// TIA Portal V19 export
VAR_GLOBAL   // PLC tag table "Digitale Ausgänge"
   A_Dkl_li_auf_CM01 AT %Q0.0 : Bool;   // Deckel links öffnen Säure CM01
   A_Dkl_li_zu_CM01 AT %Q0.1 : Bool;   // Deckel links schließen Säure CM01
   A_Dkl_re_auf_CM01 AT %Q0.2 : Bool;   // Deckel rechts öffnen Säure CM01
   A_Dkl_re_zu_CM01 AT %Q0.3 : Bool;   // Deckel rechts schließen Säure CM01
   A_Dkl_li_auf_CM02 AT %Q0.4 : Bool;   // Deckel links öffnen Säure CM02
   A_Dkl_li_zu_CM02 AT %Q0.5 : Bool;   // Deckel links schließen Säure CM02
   A_Dkl_re_auf_CM02 AT %Q0.6 : Bool;   // Deckel rechts öffnen Säure CM02
   A_Dkl_re_zu_CM02 AT %Q0.7 : Bool;   // Deckel rechts schließen Säure CM02
   "R A 1.0" AT %Q1.0 : Bool;   // Reserve
   A_LED_Q_Err AT %Q1.1 : Bool;   // LED in Taster Fehlerquittung
   A_LED_Q_NH AT %Q1.2 : Bool;   // LED in NOT-HALT Quittung
   "R A 1.3" AT %Q1.3 : Bool;   // Reserve
   "R A1.4" AT %Q1.4 : Bool;   // Turmleuchte Reserve Be-/Entladestation
   A_Mld_fertig AT %Q1.5 : Bool;   // Meldung fertig
   A_Mld_Automatik AT %Q1.6 : Bool;   // Meldung Automatik
   A_Mld_Wrn AT %Q1.7 : Bool;   // Meldung Warnung
   A_Mld_Al AT %Q2.0 : Bool;   // Meldung Störung
   A_Hupe AT %Q2.1 : Bool;   // Hupe
   A_TL_T_Vorarlarm_Gas AT %Q2.7 : Bool;   // Voralarm Gas (E13.2.)TL Tür
   A_TL_T_Hauptalarm_Gas AT %Q3.0 : Bool;   // Hauptalarm Gas (13.3) TL Tür
   A_TL_T_Hupe AT %Q3.1 : Bool;   // Hupe TL Tür
   A_KS_CM05_nicht_Voll AT %Q3.2 : Bool;   // Meldung an Wäscher Sammeltank CM05 voll
   A_KS_in_Betrieb AT %Q3.3 : Bool;   // Meldung an Wäscher und Neutralisation Säureanlage in Betrieb
   A_Mld_WS_Leckage AT %Q3.4 : Bool;   // Meldung an Werkschutz Leckage
   A_Mld_WS_Ueberlauf AT %Q3.5 : Bool;   // Meldung an Werkschutz Überlauf
   A_Mld_WS_SSt AT %Q3.6 : Bool;   // Meldung an Werkschutz Sammelstörung
   "R A 3.7" AT %Q3.7 : Bool;   // digitaler Ausgang Reserve Neutralisation
   "R A 4.0" AT %Q4.0 : Bool;   // digitaler Ausgang Reserve 1
   "R A 4.1" AT %Q4.1 : Bool;   // digitaler Ausgang Reserve 2
   "R A 4.2" AT %Q4.2 : Bool;   // digitaler Ausgang Reserve 3
   "A_Mld_fertig_Geb.G" AT %Q4.3 : Bool;   // Meldung fertig A_Mld_Automatik
   A_LED_Tuer_VS AT %Q6.0 : Bool;   // LED Tür Vorderseite CL02.SF17
   A_LED_Tuer_RS AT %Q6.1 : Bool;   // LED Tür Rückseite CL02.SF18
   A_Frg_FU_FP_HQ01 AT %Q6.2 : Bool;   // Freigabe FP HQ01 Säure CM01 CM01.GP01
   A_Frg_FU_UP_HF_CM01 AT %Q6.3 : Bool;   // Freigabe UWP Säure CM01 CM01.GP02
   A_Frg_FU_UP_H2O_CM03 AT %Q6.4 : Bool;   // Freigabe UWP Spüle CM03 CM03.GP03
   A_Frg_FU_FP_HQ02 AT %Q6.5 : Bool;   // Freigabe FP HQ02 Säure CM02 CM02.GP04
   A_Frg_FU_UP_HF_CM02 AT %Q6.6 : Bool;   // Freigabe UWP Säure CM02 CM02.GP05
   A_Frg_FU_UP_H2O_CM04 AT %Q6.7 : Bool;   // Freigabe UWP Spüle CM04 CM04.GP06
   A_Frg_FU_Vent AT %Q7.0 : Bool;   // Ventilator Ein Sperrluft FP02.GQ01
   A_RT_auf AT %Q7.1 : Bool;   // Schnelllauftor öffnen Ein-/Ausfahrt
   A_RT_zu AT %Q7.2 : Bool;   // Schnelllauftor schließen Ein-/Ausfahrt
   A_Pu_Entl_CM05 AT %Q7.3 : Bool;   // Pumpe Ein Entleerung Sammeltank CM05.GP11
   "R A 5.4" AT %Q5.4 : Bool;
   "R A 5.5" AT %Q5.5 : Bool;
   "R A 5.6" AT %Q5.6 : Bool;
   "R A 5.7" AT %Q5.7 : Bool;
   "R A 7.4" AT %Q7.4 : Bool;
   "R A 7.5" AT %Q7.5 : Bool;
   "R A 7.6" AT %Q7.6 : Bool;
   "R A 7.7" AT %Q7.7 : Bool;
   A_IBC_Vers AT %Q32.0 : Bool;   // IBC vorhanden Versorgung
   "R A 32.1" AT %Q32.1 : Bool;   // Reserve gelb Versorgung
   "R A 32.2" AT %Q32.2 : Bool;   // Reserve rot Versorgung
   "R A 32.3" AT %Q32.3 : Bool;   // Reserve Hupe Versorgung
   A_IBC_Ents AT %Q32.4 : Bool;   // IBC vorhanden Entsorgung
   "R A 32.5" AT %Q32.5 : Bool;   // Reserve gelb Versorgung
   "R A 32.6" AT %Q32.6 : Bool;   // Reserve rot Versorgung
   "R A 32.7" AT %Q32.7 : Bool;   // Reserve Hupe Versorgung
   "R A 33.0" AT %Q33.0 : Bool;
   "R A 33.1" AT %Q33.1 : Bool;
   "R A 33.2" AT %Q33.2 : Bool;
   "R A 33.3" AT %Q33.3 : Bool;
   "R A 33.4" AT %Q33.4 : Bool;
   "R A 33.5" AT %Q33.5 : Bool;
   "R A 33.6" AT %Q33.6 : Bool;
   "R A 33.7" AT %Q33.7 : Bool;
   "A_CM01.QM18" AT %Q48.0 : Bool;   // Eingang Saugleitung Filterpumpe GP01 Säure 01 CM01.QM18
   "A_CM01.QM19" AT %Q48.1 : Bool;   // Eingang Spülleitung Filterpumpe GP01 Säure 01 CM01.QM19
   "A_CM01.QM20" AT %Q48.2 : Bool;   // Eingang Spülleitung Umwälzpumpe GP02 Säure 01 CM01.QM20
   "A_HQ01.QM21" AT %Q48.4 : Bool;   // Eingang SäureleitungFiltereinheit HQ01Säure 01HQ01.QM21
   "A_HQ01.LV01" AT %Q48.3 : Bool;   // Entlüftungs-/ Überdruckventil Beutelfilter Säure 01 HQ01.LV01
   "A_HQ01.QM22" AT %Q48.5 : Bool;   // Eingang Spülleitung Filtereinheit HQ01 Säure 01 HQ01.QM22
   "A_HQ01.QM23" AT %Q48.6 : Bool;   // Ausgang Säureleitung Filtereinheit HQ01 Säure 01 HQ01.QM23
   "A_HQ01.QM24" AT %Q48.7 : Bool;   // Ausgang Spülleitung Filtereinheit HQ01 Säure 01 zu Sammeltank HQ01.QM24
   "A_CM01.QM25" AT %Q49.0 : Bool;   // Eingang Saugleitung Umwälzpumpe GP02 Säure 01 CM01.QM25
   "A_CM01.QM26" AT %Q49.1 : Bool;   // Ausgang Druckleitung Umwälzpumpe GP02 Säure 01 CM01.QM26
   "A_CM01.QM27" AT %Q49.2 : Bool;   // Ausgang Spülleitung Umwälzpumpe GP02 Säure 01 zu Sammeltank CM01.QM27
   "A_CM03.QM33" AT %Q49.3 : Bool;   // Eingang Saugleitung Umwälzpumpe GP03 Spülbecken 1 CM03.QM33
   "A_CM03.QM34" AT %Q49.4 : Bool;   // Ausgang Druckleitung Umwälzpumpe GP03 Spülbecken 1 CM03.QM34
   "A_CM03.QM36" AT %Q49.5 : Bool;   // Eingang Spülleitung Umwälzpumpe GP03 Spülbecken 1 CM03.QM36
   "A_CM03.QM37" AT %Q49.6 : Bool;   // Ausgang Spülleitung Umwälzpumpe GP03 Spülbecken 1 CM03.QM37
   "R A 49.7" AT %Q49.7 : Bool;   // Magnetventil Reserve
   "A_CM02.QM55" AT %Q50.0 : Bool;   // Eingang Saugleitung Filterpumpe GP04 Säure 02 CM02.QM55
   "A_CM02.QM56" AT %Q50.1 : Bool;   // Eingang Spülleitung Filterpumpe GP04 Säure 02 CM02.QM56
   "A_CM02.QM57" AT %Q50.2 : Bool;   // Eingang Spülleitung Umwälzpumpe GP05 Säure 02 CM02.QM57
   "A_HQ02.QM58" AT %Q50.4 : Bool;   // Eingang Spülleitung Filtereinheit HQ02 Säure 02 HQ02.QM58
   "A_HQ02.LV02" AT %Q50.3 : Bool;   // Entlüftungs-/ Überdruckventil Beutelfilter Säure 02 HQ02.LV02
   "A_HQ02.QM59" AT %Q50.5 : Bool;   // Eingang Säureleitung Filtereinheit HQ02 Säure 02 HQ02.QM59
   "A_HQ02.QM60" AT %Q50.6 : Bool;   // Ausgang Säureleitung Filtereinheit HQ02 Säure 02 HQ02.QM60
   "A_HQ02.QM61" AT %Q50.7 : Bool;   // Ausgang Spülleitung Filtereinheit HQ02 Säure 02 zu Sammeltank HQ02.QM61
   "A_CM02.QM62" AT %Q51.0 : Bool;   // Eingang Saugleitung Umwälzpumpe GP05 Säure 02 CM02.QM62
   "A_CM02.QM63" AT %Q51.1 : Bool;   // Ausgang Druckleitung Umwälzpumpe GP05 Säure 02 CM02.QM63
   "A_CM02.QM64" AT %Q51.2 : Bool;   // Ausgang Spülleitung Umwälzpumpe GP05 Säure 02 zu Sammeltank CM02.QM64
   "R A 51.3" AT %Q51.3 : Bool;   // Magnetventil Reserve
   "A_CM04.QM72" AT %Q51.4 : Bool;   // Eingang Saugleitung Umwälzpumpe GP06 Spülbecken 2 CM04.QM72
   "A_CM04.QM73" AT %Q51.5 : Bool;   // Ausgang Druckleitung Umwälzpumpe GP06 Spülbecken 2 CM04.QM73
   "A_CM04.QM75" AT %Q51.6 : Bool;   // Eingang Spülleitung Umwälzpumpe GP06 Spülbecken 2 CM04.QM75
   "R A 51.7" AT %Q51.7 : Bool;   // Magnetventil Reserve
   "A_CM04.QM76" AT %Q52.0 : Bool;   // Ausgang Spülleitung Umwälzpumpe GP06 Spülbecken 2 CM04.QM76
   "A_CM04.QM77" AT %Q52.1 : Bool;   // Frischwasserzufuhr Nachdosierung Spülbecken 2 CM04.QM77
   "A_CL01.GP08" AT %Q52.2 : Bool;   // Membranpumpe GP08 Sumpfentleerung Übergabestation CL01.GP08
   "A_CL02.GP09" AT %Q52.3 : Bool;   // Membranpumpe GP09 Sumpfentleerung Säurebecken CL02.GP09
   "A_CL01.QM51" AT %Q52.4 : Bool;   // Zuleitung VE-Wasser-Spülung Pumpe GP08 CL01.QM51
   "A_CL02.QM52" AT %Q52.5 : Bool;   // Zuleitung VE-Wasser-Spülung Pumpe GP09 CL01.QM52
   "R A 52.6" AT %Q52.6 : Bool;   // Magnetventil Reserve
   "R A 52.7" AT %Q52.7 : Bool;   // Magnetventil Reserve
   "A_CM05.QM61" AT %Q53.0 : Bool;   // Saugseite Förderpumpe Entleerung GP11 Sammeltank CM05 CM05.QM61
   "A_CM05.QM62" AT %Q53.1 : Bool;   // Eingang Spülleitung Förderpumpe GP11 Sammeltank CM05 CM05.QM62
   "A_CM05.QM63" AT %Q53.2 : Bool;   // Ausgang Spülleitung Förderpumpe GP11 Sammeltank CM05 CM05.QM63
   "A_CM05.QM64" AT %Q53.3 : Bool;   // Druckseite Förderpumpe Entleerung GP11 Sammeltank CM05 CM05.QM64
   "R A 53.4" AT %Q53.4 : Bool;   // Magnetventil Reserve
   "R A 53.5" AT %Q53.5 : Bool;   // Magnetventil Reserve
   "R A 53.6" AT %Q53.6 : Bool;   // Magnetventil Reserve
   "R A 53.7" AT %Q53.7 : Bool;   // Magnetventil Reserve
   "A_CM03.QM35" AT %Q64.0 : Bool;   // VE-Wasserleitung Spritzregister Spülbecken 1 CM03.QM35
   "A_CM04.QM74" AT %Q64.1 : Bool;   // VE-Wasserleitung Spritzregister Spülbecken 2 CM04.QM74
   "A_GP01.GP12" AT %Q64.2 : Bool;   // Druckluftmembran- Leckagepumpe GP12 Versorgung Frischsäure GP01.GP12
   "A_GP01.GP13" AT %Q64.3 : Bool;   // Druckluftmembran- pumpe GP13 Versorgung Frischsäure GP01.GP13
   "A_GP01.QM14" AT %Q64.4 : Bool;   // PFA Schlauchleitung Anbindung IBC Quick Connect Entsorgung GP01.QM14
   "A_GP01.QM15" AT %Q64.5 : Bool;   // Eingang Saugleitung Membranpumpe GP13 Versorgung Frischsäure GP01.QM15
   "A_GP01.QM16" AT %Q64.6 : Bool;   // Eingang Spülleitung Membranpumpe GP13 Versorgung Frischsäure GP01.QM16
   "A_GP01.QM17" AT %Q64.7 : Bool;   // Ausgang Spülleitung Membranpumpe GP13 Versorgung zu Sammeltank GP01.QM17
   "A_GP01.QM18" AT %Q65.0 : Bool;   // Ausgang Druckleitung Membranpumpe GP13 Versorgung zu UV-GP01 GP01.QM18
   "A_GP01.QM19" AT %Q65.1 : Bool;   // Verriegelung UV-GP01 Versorgungsleitung zu Säure CM02 GP01.QM19
   "A_GP01.QM20" AT %Q65.2 : Bool;   // Verriegelung UV-GP01 Versorgungsleitung zu Säure CM01 GP01.QM20
   "A_GP01.QM21" AT %Q65.3 : Bool;   // Verriegelung UV-GP01 Versorgungsleitung zur Entsorgung GP02 GP01.QM21
   "A_GP01.QM22" AT %Q65.4 : Bool;   // Verriegelung UV-GP01 Versorgungsleitung zur Versorgung GP01 GP01.QM22
   "A_GP01.QM23" AT %Q65.5 : Bool;   // VE-Wasser-Spülung GP12 zu Auffangwanne GP01.QM23
   "A_GP02.GP07" AT %Q65.6 : Bool;   // Druckluftmembran- Leckagepumpe GP07 Entsorgung Altsäure GP02.GP07
   "A_GP02.GP10" AT %Q65.7 : Bool;   // Druckluftmembran- pumpe GP10 Versorgung aus GP02 GP02.GP10
   "A_GP02.QM37" AT %Q66.0 : Bool;   // VE-Wasser-Ventil Leckagesumpf Entsorgung Altsäure GP02.QM37
   "A_GP02.QM38" AT %Q66.1 : Bool;   // Eingang Saugleitung Membranpumpe GP10 Versorgung aus GP02 GP02.QM38
   "A_GP02.QM39" AT %Q66.2 : Bool;   // Eingang Spülleitung Membranpumpe GP10 Versorgung aus GP02 GP02.QM39
   "A_GP02.QM40" AT %Q66.3 : Bool;   // Ausgang Spülleitung Membranpumpe GP10 zu Sammeltank CM05 GP02.QM40
   "A_GP02.QM41" AT %Q66.4 : Bool;   // Verriegelung UV-GP02 Entsorgungsleitung zu UV-GP02 GP02.QM41
   "A_GP02.QM42" AT %Q66.5 : Bool;   // Ausgang Spülleitung Membranpumpe GP10 zu Sammeltank CM05 GP02.QM42
   "A_GP02.QM43" AT %Q66.6 : Bool;   // Verriegelung UV-GP02 Entsorgungsleitung zu Entsorgung GP02 GP02.QM43
   "A_GP02.QM44" AT %Q66.7 : Bool;   // Verriegelung UV-GP02 Entsorgungsleitung zu Versorgung GP01 GP02.QM44
   "A_GP02.QM45" AT %Q67.0 : Bool;   // Verriegelung UV-GP02 Entsorgungsleitung von Säurebecken CM01 GP02.QM45
   "A_GP02.QM46" AT %Q67.1 : Bool;   // Verriegelung UV-GP02 Entsorgungsleitung von Säurebecken CM02 GP02.QM46
   "A_CM05.GP14" AT %Q67.2 : Bool;   // Membranpumpe GP14 Entleerung Becken CM01-CM04 CM05.GP14
   "R A 67.3" AT %Q67.3 : Bool;   // Magnetventil Reserve
   "R A 67.4" AT %Q67.4 : Bool;   // Magnetventil Reserve
   "R A 67.5" AT %Q67.5 : Bool;   // Magnetventil Reserve
   "R A 67.6" AT %Q67.6 : Bool;   // Magnetventil Reserve
   "R A 67.7" AT %Q67.7 : Bool;   // Magnetventil Reserve
   "A_Mld_Automatik_Geb.G" AT %Q4.4 : Bool;   // Meldung Automatik Gebäude G
   "A_Mld_Wrn_Geb.G" AT %Q4.5 : Bool;   // Meldung Warnung Gebäude G
   "A_Mld_Al_Geb.G" AT %Q4.6 : Bool;   // Meldung Störung Gebäude G
   "A_Hupe_Geb.G" AT %Q4.7 : Bool;   // Meldung Hupe Gebäude G
   "A_TL_T_Vorarlarm_Gas(2)" AT %Q5.0 : Bool;   // Voralarm Gas (E13.2.)TL Tür
   "A_TL_T_Hauptalarm_Gas(2)" AT %Q5.1 : Bool;   // Hauptalarm Gas (E13.3) TL Tür
   "A_TL_T_Hupe(2)" AT %Q5.2 : Bool;   // Hupe TL Tür
   "R A 5.3" AT %Q5.3 : Bool;
   "A_Mld_fertig(2)" AT %Q2.2 : Bool;   // Meldung fertig
   "A_Mld_Automatik(2)" AT %Q2.3 : Bool;   // Meldung Automatik
   "A_Mld_Wrn(2)" AT %Q2.4 : Bool;   // Meldung Warnung
   "A_Mld_Al(2)" AT %Q2.5 : Bool;   // Meldung Störung
   "A_Hupe(2)" AT %Q2.6 : Bool;   // Hupe
   A_Frg_FU_QF_WR02 AT %Q72.0 : Bool;   // Freigabe Querumsetzer WR02
   A_Frg_FU_QF_WR03 AT %Q72.1 : Bool;   // Freigabe Querumsetzer WR03
   "R A 72.2" AT %Q72.2 : Bool;
   "R A 72.3" AT %Q72.3 : Bool;
   "R A 72.4" AT %Q72.4 : Bool;
   "R A 72.5" AT %Q72.5 : Bool;
   "R A 72.6" AT %Q72.6 : Bool;
   "R A 72.7" AT %Q72.7 : Bool;
   A_Hupe_QF AT %Q73.0 : Bool;   // Hupe
   "R A 73.1" AT %Q73.1 : Bool;
   "R A 73.2" AT %Q73.2 : Bool;
   "R A 73.3" AT %Q73.3 : Bool;
   "R A 73.4" AT %Q73.4 : Bool;
   "R A 73.5" AT %Q73.5 : Bool;
   "R A 73.6" AT %Q73.6 : Bool;
   "R A 73.7" AT %Q73.7 : Bool;
   A_RepB AT %Q80.0 : Bool;   // Reparaturbetrieb Manipulator WR04, WR05
   A_Snk_re AT %Q80.1 : Bool;   // senken Hubwerk rechts Manipulator WR04
   A_Heb_re AT %Q80.2 : Bool;   // heben Hubwerk rechts Manipulator WR04
   A_Snk_li AT %Q80.3 : Bool;   // Senken Hubwerk links Manipulator WR05
   A_Heb_li AT %Q80.4 : Bool;   // Heben Hubwerk links Manipulator WR05
   A_Frg_FU_Fahrt AT %Q80.5 : Bool;   // Freigabe Kranfahrwerk Manipulator
   A_Frg_FU_Hub_re AT %Q80.6 : Bool;   // Freigabe Hubwerk rechts Manipulator
   A_WZ_Tara_re_1 AT %Q80.7 : Bool;   // Hubwerk rechts Wägezelle 1 Tara WR04.BW01
   A_WZ_Tara_re_2 AT %Q81.0 : Bool;   // Hubwerk rechts Wägezelle 2 Tara WR04.BW02
   A_WZ_Tara_re_3 AT %Q81.1 : Bool;   // Hubwerk rechts Wägezelle 3 Tara WR04.BW03
   A_WZ_Tara_re_4 AT %Q81.2 : Bool;   // Hubwerk rechts Wägezelle 4 Tara WR04.BW04
   A_Frg_FU_Hub_li AT %Q81.3 : Bool;   // Freigabe Hubwerk links Manipulator
   A_WZ_Tara_li_1 AT %Q81.4 : Bool;   // Hubwerk links Wägezelle 1 Tara WR05.BW01
   A_WZ_Tara_li_2 AT %Q81.5 : Bool;   // Hubwerk links Wägezelle 2 Tara WR05.BW02
   A_WZ_Tara_li_3 AT %Q81.6 : Bool;   // Hubwerk links Wägezelle 3 Tara WR05.BW03
   A_WZ_Tara_li_4 AT %Q81.7 : Bool;   // Hubwerk links Wägezelle 4 Tara WR05.BW04
   AW_Steuer_348i_TW1 AT %QW314 : Word;   // Steuerwort Laser TW1
   AD_Preset_SL_Hub_links AT %QD321 : DInt;
   AD_Preset_SL_Hub_rechts AT %QD331 : DWord;
   AB_StB_Preset_SL_Hub_links AT %QB320 : Byte;
   AB_StB_Preset_SL_Hub_rechts AT %QB330 : Byte;
   A_Preset_SL_Hub_links AT %Q320.0 : Bool;
   A_Preset_SL_Hub_rechts AT %Q330.0 : Bool;
END_VAR
